TYPE CHECK_EOF_ACTION EXTENDS FILE_ACTION :
STRUCT
	Callback : ICheckEofActionCallback;
END_STRUCT
END_TYPE

(* stored: Version 1.1.0.1
   DUT CHECK_EOF_ACTION: Id {601f2068-92c9-4f41-ba11-2041fa10ea62} *)
